FUNCTION_BLOCK FB_Area
VAR
	name : STRING; //fully area name
	id : INT; //area number only
	
	queue : PtrQueue := (dataSize := SIZEOF(POINTER TO Bundle));
	activeBundles : ARRAY[0..10] OF Bundle; //most will only use 1
	capacity : USINT;
	
	ready : BOOL; //ready to receive
	done : BOOL; //finished current bundle new bundle
	
	socket : AdsSocket;
END_VAR
VAR CONSTANT
	test : INT;
END_VAR

METHOD transfer : BOOL
VAR_INPUT
END_VAR
END_METHOD

END_FUNCTION_BLOCK

(* stored: Version 1.1.0.1, ProductVersion 3.1.4024.11
   POU FB_Area: Id {cd10b598-7a8c-4b57-8c3c-62834945eee3}, SpecialFunc None
   Method transfer: Id {6890ed38-c4b0-403c-9342-b4dcfc2d0725} *)
